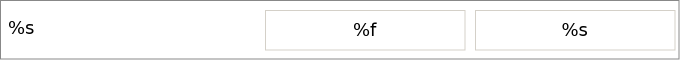
VISUALIZATION SingleRecipesParameterTypeReal  // 680x60
VAR_IN_OUT
	stRecipeParameter : ST_VisuCtrlRecipeParameter;
END_VAR
    Textfield (265,10 200x40), "%f", text variable: stRecipeParameter.rValue
        OnMouseClick: write the text variable via VisuDialogs.Numpad
    Textfield (475,10 200x40), "%s", text variable: stRecipeParameter.sFileValue
    Textfield (5,8 250x40), "%s", text variable: stRecipeParameter.sName
END_VISUALIZATION

(* stored: Version 1.1.0.1, ProductVersion 3.1.4024.12
   Visu SingleRecipesParameterTypeReal: Id {b70dd14f-eff8-4c55-93b4-8d15366832cd} *)
